(* IEC 61131-3 sources: CodesysTest/alpha/export/Device.dev/Plc Logic/Application/FBs/FB_FaultHandler.pou, 1 file *)

(* ---- registerFaultSource.m.st ---- *)
(*#-#-#-#-#-#-#-#-#-#---Declaration---#-#-#-#-#-#-#-#-#-#-#-#-#*)

METHOD registerFaultSource
VAR_INPUT
     faultSource : REFERENCE TO IFault;
END_VAR

(*#-#-#-#-#-#-#-#-#-#---Implementation---#-#-#-#-#-#-#-#-#-#-#-#-#*)

faultSourceList[sourcesInList]:= faultSource;
sourcesInList:= sourcesInList + 1;
